// TIA Portal V18 export
ORGANIZATION_BLOCK "Safety"   // OB126, LAD, ProgramCycle
TITLE = "Main Program Sweep (Cycle)"
{ S7_Optimized_Access := 'TRUE' }
VERSION : 0.1
// stored: AutoNumber true, IsIECCheckEnabled false, SetENOAutomatically false
   VAR_INPUT
      Initial_Call : Bool;   // Initial call of this OB
      Remanence : Bool;   // =True, if remanent data are available
   END_VAR
   VAR_TEMP
      FaultReset : Bool;
      bRetVal : Int;
   END_VAR
   VAR_TEMP   // added for the SCL form of the ladder/FBD networks
      _w1 : Bool;
      _w2 : Bool;
      _w3 : Bool;
   END_VAR
BEGIN

REGION Network 1: ESTOP Release Edge
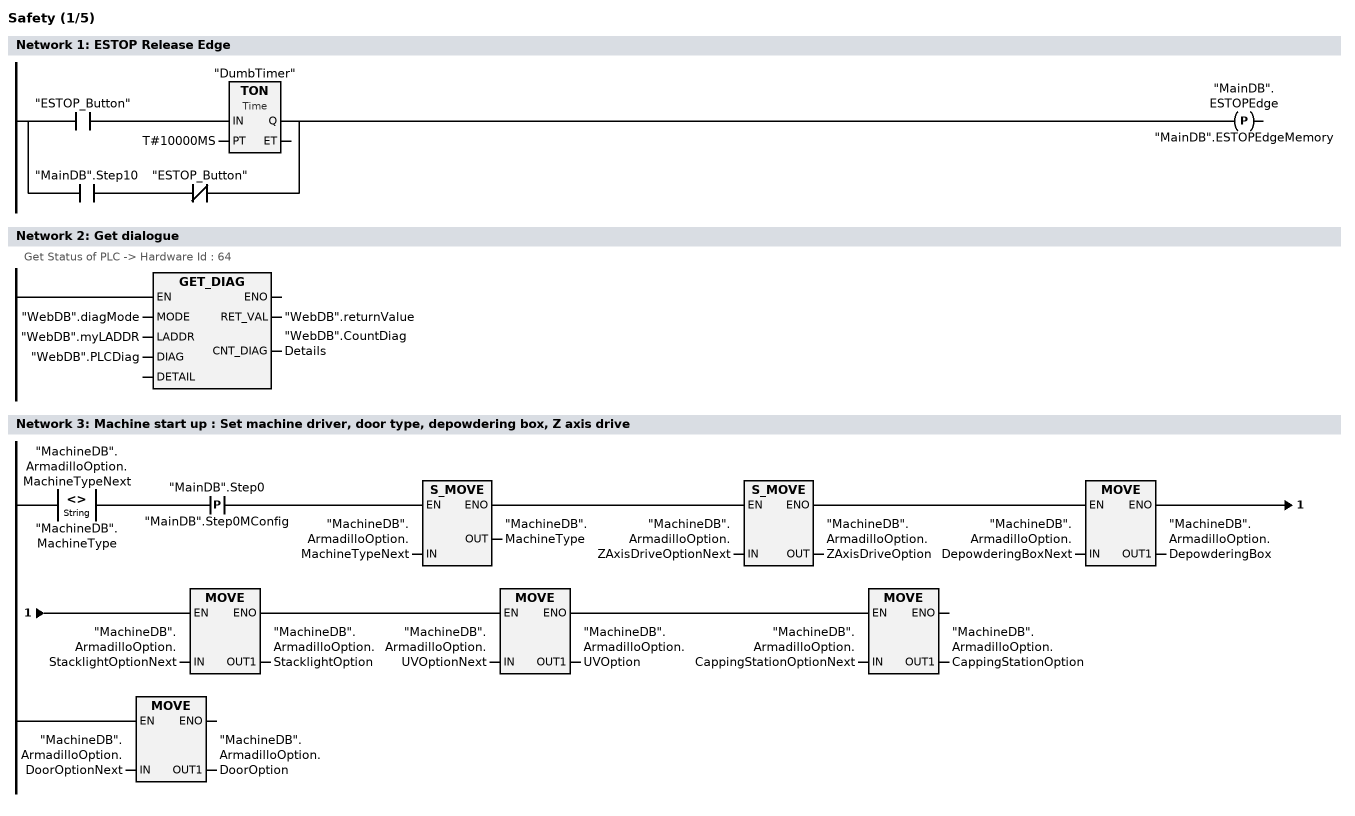
   "DumbTimer".TON(IN := "ESTOP_Button", PT := T#10000MS);
   #_w1 := "DumbTimer".Q OR ("MainDB".Step10 AND NOT "ESTOP_Button");
   "MainDB".ESTOPEdge := #_w1 AND NOT "MainDB".ESTOPEdgeMemory;   // rising edge
   "MainDB".ESTOPEdgeMemory := #_w1;
END_REGION

REGION Network 2: Get dialogue
   // Get Status of PLC -> Hardware Id : 64
   RUNG wire#powerrail
      GET_DIAG(MODE := "WebDB".diagMode, LADDR := "WebDB".myLADDR, DIAG := "WebDB".PLCDiag, DETAIL :=, RET_VAL => "WebDB".returnValue, CNT_DIAG => "WebDB".CountDiagDetails)
   END_RUNG
   // the same network as SCL:
   "WebDB".returnValue := GET_DIAG(MODE := "WebDB".diagMode,
                           LADDR := "WebDB".myLADDR,
                           DIAG := "WebDB".PLCDiag,
                           CNT_DIAG => "WebDB".CountDiagDetails);
END_REGION

REGION Network 3: Machine start up : Set machine driver, door type, depowdering box, Z axis drive
   RUNG wire#powerrail
      { S7_Templates := "SrcType := String" } NE_Contact(in1 := "MachineDB".ArmadilloOption.MachineTypeNext, in2 := "MachineDB".MachineType)
      P_Contact(operand := "MainDB".Step0, bit := "MainDB".Step0MConfig)
      S_Move(in := "MachineDB".ArmadilloOption.MachineTypeNext, out => "MachineDB".MachineType)
      S_Move(in := "MachineDB".ArmadilloOption.ZAxisDriveOptionNext, out => "MachineDB".ArmadilloOption.ZAxisDriveOption)
      Move(in := "MachineDB".ArmadilloOption.DepowderingBoxNext, out1 => "MachineDB".ArmadilloOption.DepowderingBox)
      Move(in := "MachineDB".ArmadilloOption.StacklightOptionNext, out1 => "MachineDB".ArmadilloOption.StacklightOption)
      Move(in := "MachineDB".ArmadilloOption.UVOptionNext, out1 => "MachineDB".ArmadilloOption.UVOption)
      Move(in := "MachineDB".ArmadilloOption.CappingStationOptionNext, out1 => "MachineDB".ArmadilloOption.CappingStationOption)
   END_RUNG
   RUNG wire#powerrail
      Move(in := "MachineDB".ArmadilloOption.DoorOptionNext, out1 => "MachineDB".ArmadilloOption.DoorOption)
   END_RUNG
   // the same network as SCL:
   #_w1 := ("MachineDB".ArmadilloOption.MachineTypeNext <> "MachineDB".MachineType) AND "MainDB".Step0 AND NOT "MainDB".Step0MConfig;   // rising edge of "MainDB".Step0
   "MainDB".Step0MConfig := "MainDB".Step0;
   IF #_w1 THEN
       "MachineDB".MachineType := "MachineDB".ArmadilloOption.MachineTypeNext;
       "MachineDB".ArmadilloOption.ZAxisDriveOption := "MachineDB".ArmadilloOption.ZAxisDriveOptionNext;
       "MachineDB".ArmadilloOption.DepowderingBox := "MachineDB".ArmadilloOption.DepowderingBoxNext;
       "MachineDB".ArmadilloOption.StacklightOption := "MachineDB".ArmadilloOption.StacklightOptionNext;
       "MachineDB".ArmadilloOption.UVOption := "MachineDB".ArmadilloOption.UVOptionNext;
       "MachineDB".ArmadilloOption.CappingStationOption := "MachineDB".ArmadilloOption.CappingStationOptionNext;
   END_IF;
   "MachineDB".ArmadilloOption.DoorOption := "MachineDB".ArmadilloOption.DoorOptionNext;
END_REGION

REGION Network 4: MachineDriverSettingArray
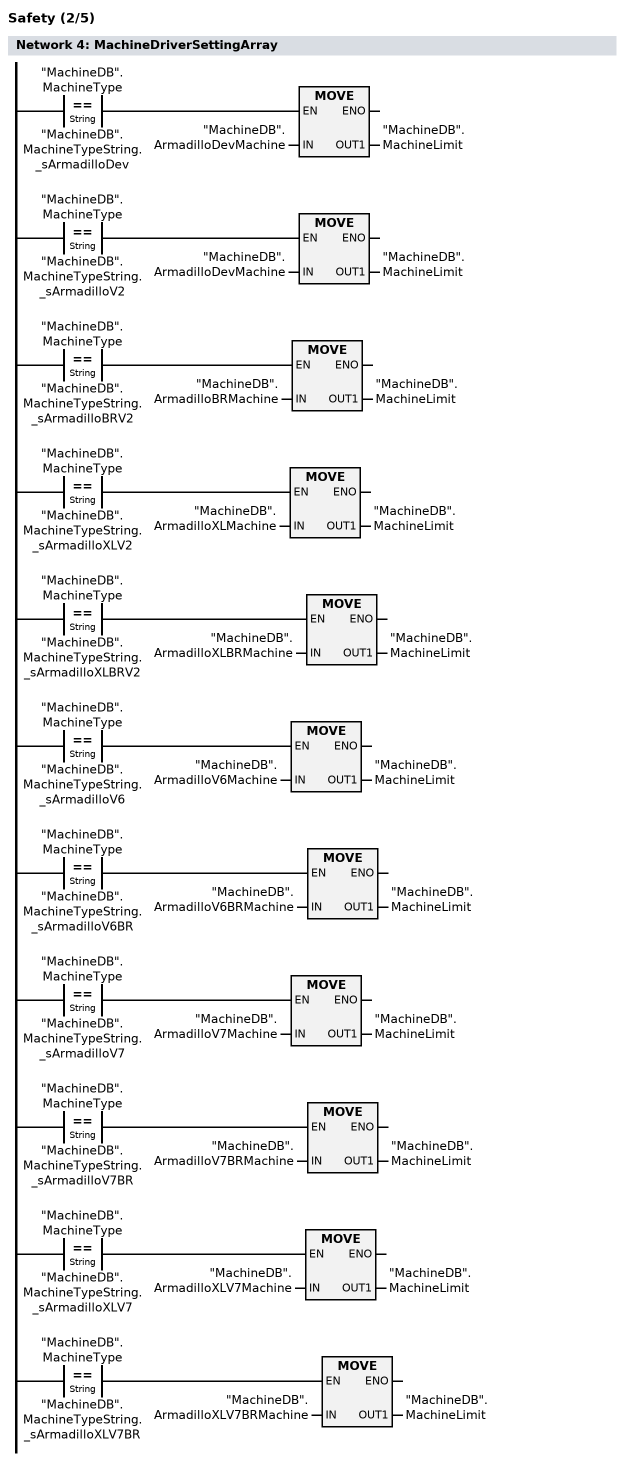
   RUNG wire#powerrail
      { S7_Templates := "SrcType := String" } EQ_Contact(in1 := "MachineDB".MachineType, in2 := "MachineDB".MachineTypeString._sArmadilloDev)
      Move(in := "MachineDB".ArmadilloDevMachine, out1 => "MachineDB".MachineLimit)
   END_RUNG
   RUNG wire#powerrail
      { S7_Templates := "SrcType := String" } EQ_Contact(in1 := "MachineDB".MachineType, in2 := "MachineDB".MachineTypeString._sArmadilloV2)
      Move(in := "MachineDB".ArmadilloDevMachine, out1 => "MachineDB".MachineLimit)
   END_RUNG
   RUNG wire#powerrail
      { S7_Templates := "SrcType := String" } EQ_Contact(in1 := "MachineDB".MachineType, in2 := "MachineDB".MachineTypeString._sArmadilloBRV2)
      Move(in := "MachineDB".ArmadilloBRMachine, out1 => "MachineDB".MachineLimit)
   END_RUNG
   RUNG wire#powerrail
      { S7_Templates := "SrcType := String" } EQ_Contact(in1 := "MachineDB".MachineType, in2 := "MachineDB".MachineTypeString._sArmadilloXLV2)
      Move(in := "MachineDB".ArmadilloXLMachine, out1 => "MachineDB".MachineLimit)
   END_RUNG
   RUNG wire#powerrail
      { S7_Templates := "SrcType := String" } EQ_Contact(in1 := "MachineDB".MachineType, in2 := "MachineDB".MachineTypeString._sArmadilloXLBRV2)
      Move(in := "MachineDB".ArmadilloXLBRMachine, out1 => "MachineDB".MachineLimit)
   END_RUNG
   RUNG wire#powerrail
      { S7_Templates := "SrcType := String" } EQ_Contact(in1 := "MachineDB".MachineType, in2 := "MachineDB".MachineTypeString._sArmadilloV6)
      Move(in := "MachineDB".ArmadilloV6Machine, out1 => "MachineDB".MachineLimit)
   END_RUNG
   RUNG wire#powerrail
      { S7_Templates := "SrcType := String" } EQ_Contact(in1 := "MachineDB".MachineType, in2 := "MachineDB".MachineTypeString._sArmadilloV6BR)
      Move(in := "MachineDB".ArmadilloV6BRMachine, out1 => "MachineDB".MachineLimit)
   END_RUNG
   RUNG wire#powerrail
      { S7_Templates := "SrcType := String" } EQ_Contact(in1 := "MachineDB".MachineType, in2 := "MachineDB".MachineTypeString._sArmadilloV7)
      Move(in := "MachineDB".ArmadilloV7Machine, out1 => "MachineDB".MachineLimit)
   END_RUNG
   RUNG wire#powerrail
      { S7_Templates := "SrcType := String" } EQ_Contact(in1 := "MachineDB".MachineType, in2 := "MachineDB".MachineTypeString._sArmadilloV7BR)
      Move(in := "MachineDB".ArmadilloV7BRMachine, out1 => "MachineDB".MachineLimit)
   END_RUNG
   RUNG wire#powerrail
      { S7_Templates := "SrcType := String" } EQ_Contact(in1 := "MachineDB".MachineType, in2 := "MachineDB".MachineTypeString._sArmadilloXLV7)
      Move(in := "MachineDB".ArmadilloXLV7Machine, out1 => "MachineDB".MachineLimit)
   END_RUNG
   RUNG wire#powerrail
      { S7_Templates := "SrcType := String" } EQ_Contact(in1 := "MachineDB".MachineType, in2 := "MachineDB".MachineTypeString._sArmadilloXLV7BR)
      Move(in := "MachineDB".ArmadilloXLV7BRMachine, out1 => "MachineDB".MachineLimit)
   END_RUNG
   // the same network as SCL:
   IF "MachineDB".MachineType = "MachineDB".MachineTypeString._sArmadilloDev THEN
       "MachineDB".MachineLimit := "MachineDB".ArmadilloDevMachine;
   END_IF;
   IF "MachineDB".MachineType = "MachineDB".MachineTypeString._sArmadilloV2 THEN
       "MachineDB".MachineLimit := "MachineDB".ArmadilloDevMachine;
   END_IF;
   IF "MachineDB".MachineType = "MachineDB".MachineTypeString._sArmadilloBRV2 THEN
       "MachineDB".MachineLimit := "MachineDB".ArmadilloBRMachine;
   END_IF;
   IF "MachineDB".MachineType = "MachineDB".MachineTypeString._sArmadilloXLV2 THEN
       "MachineDB".MachineLimit := "MachineDB".ArmadilloXLMachine;
   END_IF;
   IF "MachineDB".MachineType = "MachineDB".MachineTypeString._sArmadilloXLBRV2 THEN
       "MachineDB".MachineLimit := "MachineDB".ArmadilloXLBRMachine;
   END_IF;
   IF "MachineDB".MachineType = "MachineDB".MachineTypeString._sArmadilloV6 THEN
       "MachineDB".MachineLimit := "MachineDB".ArmadilloV6Machine;
   END_IF;
   IF "MachineDB".MachineType = "MachineDB".MachineTypeString._sArmadilloV6BR THEN
       "MachineDB".MachineLimit := "MachineDB".ArmadilloV6BRMachine;
   END_IF;
   IF "MachineDB".MachineType = "MachineDB".MachineTypeString._sArmadilloV7 THEN
       "MachineDB".MachineLimit := "MachineDB".ArmadilloV7Machine;
   END_IF;
   IF "MachineDB".MachineType = "MachineDB".MachineTypeString._sArmadilloV7BR THEN
       "MachineDB".MachineLimit := "MachineDB".ArmadilloV7BRMachine;
   END_IF;
   IF "MachineDB".MachineType = "MachineDB".MachineTypeString._sArmadilloXLV7 THEN
       "MachineDB".MachineLimit := "MachineDB".ArmadilloXLV7Machine;
   END_IF;
   IF "MachineDB".MachineType = "MachineDB".MachineTypeString._sArmadilloXLV7BR THEN
       "MachineDB".MachineLimit := "MachineDB".ArmadilloXLV7BRMachine;
   END_IF;
END_REGION

REGION Network 5: No Go Zone 01
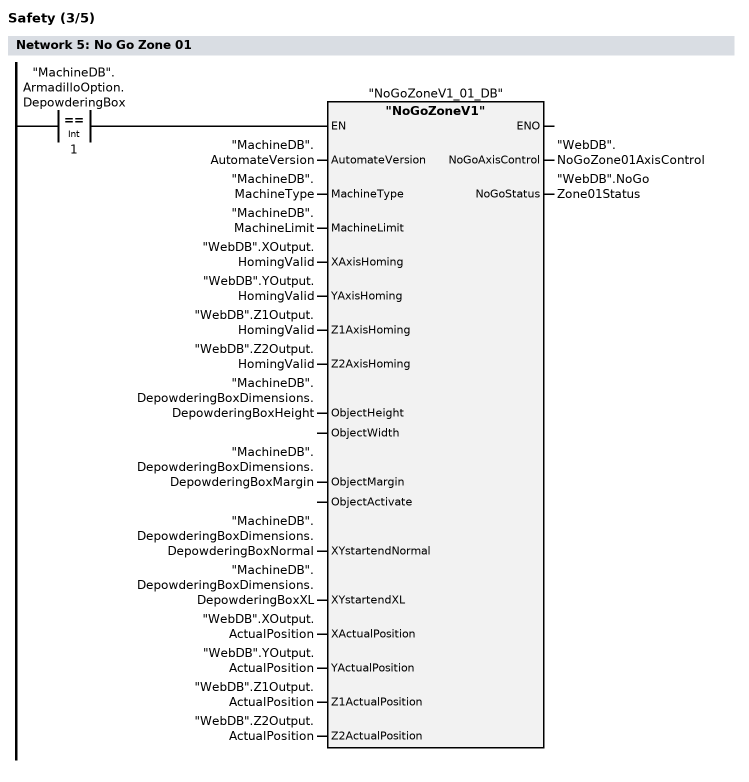
   RUNG wire#powerrail
      { S7_Templates := "SrcType := Int" } EQ_Contact(in1 := "MachineDB".ArmadilloOption.DepowderingBox, in2 := 1)
      "NoGoZoneV1_01_DB"(AutomateVersion := "MachineDB".AutomateVersion, MachineType := "MachineDB".MachineType, MachineLimit := "MachineDB".MachineLimit, XAxisHoming := "WebDB".XOutput.HomingValid, YAxisHoming := "WebDB".YOutput.HomingValid, Z1AxisHoming := "WebDB".Z1Output.HomingValid, Z2AxisHoming := "WebDB".Z2Output.HomingValid, ObjectHeight := "MachineDB".DepowderingBoxDimensions.DepowderingBoxHeight, ObjectWidth :=, ObjectMargin := "MachineDB".DepowderingBoxDimensions.DepowderingBoxMargin, ObjectActivate :=, XYstartendNormal := "MachineDB".DepowderingBoxDimensions.DepowderingBoxNormal, XYstartendXL := "MachineDB".DepowderingBoxDimensions.DepowderingBoxXL, XActualPosition := "WebDB".XOutput.ActualPosition, YActualPosition := "WebDB".YOutput.ActualPosition, Z1ActualPosition := "WebDB".Z1Output.ActualPosition, Z2ActualPosition := "WebDB".Z2Output.ActualPosition, NoGoAxisControl => "WebDB".NoGoZone01AxisControl, NoGoStatus => "WebDB".NoGoZone01Status)
   END_RUNG
   // the same network as SCL:
   IF "MachineDB".ArmadilloOption.DepowderingBox = 1 THEN
       "NoGoZoneV1_01_DB"(AutomateVersion := "MachineDB".AutomateVersion,   // "NoGoZoneV1"
                          MachineType := "MachineDB".MachineType,
                          MachineLimit := "MachineDB".MachineLimit,
                          XAxisHoming := "WebDB".XOutput.HomingValid,
                          YAxisHoming := "WebDB".YOutput.HomingValid,
                          Z1AxisHoming := "WebDB".Z1Output.HomingValid,
                          Z2AxisHoming := "WebDB".Z2Output.HomingValid,
                          ObjectHeight := "MachineDB".DepowderingBoxDimensions.DepowderingBoxHeight,
                          ObjectMargin := "MachineDB".DepowderingBoxDimensions.DepowderingBoxMargin,
                          XYstartendNormal := "MachineDB".DepowderingBoxDimensions.DepowderingBoxNormal,
                          XYstartendXL := "MachineDB".DepowderingBoxDimensions.DepowderingBoxXL,
                          XActualPosition := "WebDB".XOutput.ActualPosition,
                          YActualPosition := "WebDB".YOutput.ActualPosition,
                          Z1ActualPosition := "WebDB".Z1Output.ActualPosition,
                          Z2ActualPosition := "WebDB".Z2Output.ActualPosition,
                          NoGoAxisControl => "WebDB".NoGoZone01AxisControl,
                          NoGoStatus => "WebDB".NoGoZone01Status);
   END_IF;
END_REGION

REGION Network 6: Door Sensor
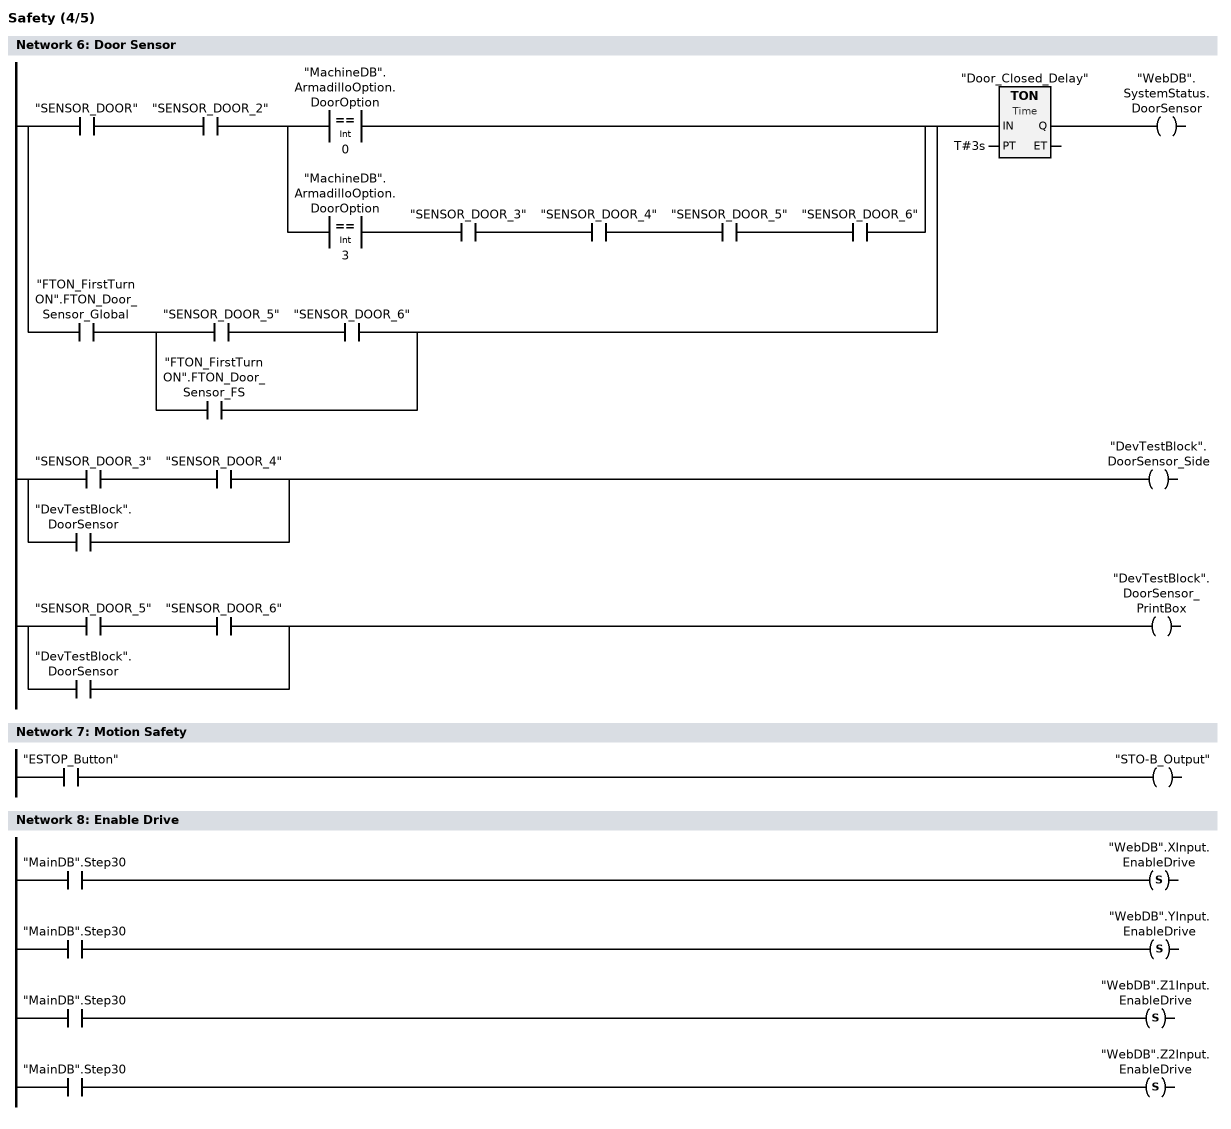
   RUNG wire#powerrail
      Contact( "SENSOR_DOOR" )
      Contact( "SENSOR_DOOR_2" )
      wire#w1
      { S7_Templates := "SrcType := Int" } EQ_Contact(in1 := "MachineDB".ArmadilloOption.DoorOption, in2 := 0)
      wire#w2
      { S7_Templates := "time_type := Time" } "Door_Closed_Delay".TON(pt := T#3s, et =>)
      Coil( "WebDB".SystemStatus.DoorSensor )
   END_RUNG
   RUNG wire#w1
      { S7_Templates := "SrcType := Int" } EQ_Contact(in1 := "MachineDB".ArmadilloOption.DoorOption, in2 := 3)
      Contact( "SENSOR_DOOR_3" )
      Contact( "SENSOR_DOOR_4" )
      Contact( "SENSOR_DOOR_5" )
      Contact( "SENSOR_DOOR_6" )
   END_RUNG wire#w2
   RUNG wire#powerrail
      Contact( "FTON_FirstTurnON".FTON_Door_Sensor_Global )
      wire#w3
      Contact( "SENSOR_DOOR_5" )
      Contact( "SENSOR_DOOR_6" )
   END_RUNG wire#w2
   RUNG wire#w3
      Contact( "FTON_FirstTurnON".FTON_Door_Sensor_FS )
   END_RUNG wire#w2
   RUNG wire#powerrail
      Contact( "SENSOR_DOOR_3" )
      Contact( "SENSOR_DOOR_4" )
      wire#w4
      Coil( "DevTestBlock".DoorSensor_Side )
   END_RUNG
   RUNG wire#powerrail
      Contact( "DevTestBlock".DoorSensor )
   END_RUNG wire#w4
   RUNG wire#powerrail
      Contact( "SENSOR_DOOR_5" )
      Contact( "SENSOR_DOOR_6" )
      wire#w5
      Coil( "DevTestBlock".DoorSensor_PrintBox )
   END_RUNG
   RUNG wire#powerrail
      Contact( "DevTestBlock".DoorSensor )
   END_RUNG wire#w5
   // the same network as SCL:
   "Door_Closed_Delay".TON(IN := ("SENSOR_DOOR" AND "SENSOR_DOOR_2" AND (("MachineDB".ArmadilloOption.DoorOption = 0) OR (("MachineDB".ArmadilloOption.DoorOption = 3) AND "SENSOR_DOOR_3" AND "SENSOR_DOOR_4" AND "SENSOR_DOOR_5" AND "SENSOR_DOOR_6"))) OR ("FTON_FirstTurnON".FTON_Door_Sensor_Global AND (("SENSOR_DOOR_5" AND "SENSOR_DOOR_6") OR "FTON_FirstTurnON".FTON_Door_Sensor_FS)),
                           PT := T#3s);
   "WebDB".SystemStatus.DoorSensor := "Door_Closed_Delay".Q;
   "DevTestBlock".DoorSensor_Side := ("SENSOR_DOOR_3" AND "SENSOR_DOOR_4") OR "DevTestBlock".DoorSensor;
   "DevTestBlock".DoorSensor_PrintBox := ("SENSOR_DOOR_5" AND "SENSOR_DOOR_6") OR "DevTestBlock".DoorSensor;
END_REGION

REGION Network 7: Motion Safety
   RUNG wire#powerrail
      Contact( "ESTOP_Button" )
      Coil( "STO-B_Output" )
   END_RUNG
   // the same network as SCL:
   "STO-B_Output" := "ESTOP_Button";
END_REGION

REGION Network 8: Enable Drive
   RUNG wire#powerrail
      Contact( "MainDB".Step30 )
      S_Coil( "WebDB".XInput.EnableDrive )
   END_RUNG
   RUNG wire#powerrail
      Contact( "MainDB".Step30 )
      S_Coil( "WebDB".YInput.EnableDrive )
   END_RUNG
   RUNG wire#powerrail
      Contact( "MainDB".Step30 )
      S_Coil( "WebDB".Z1Input.EnableDrive )
   END_RUNG
   RUNG wire#powerrail
      Contact( "MainDB".Step30 )
      S_Coil( "WebDB".Z2Input.EnableDrive )
   END_RUNG
   // the same network as SCL:
   IF "MainDB".Step30 THEN
       "WebDB".XInput.EnableDrive := TRUE;
       "WebDB".YInput.EnableDrive := TRUE;
       "WebDB".Z1Input.EnableDrive := TRUE;
       "WebDB".Z2Input.EnableDrive := TRUE;
   END_IF;
END_REGION

REGION Network 9: Disable Drive
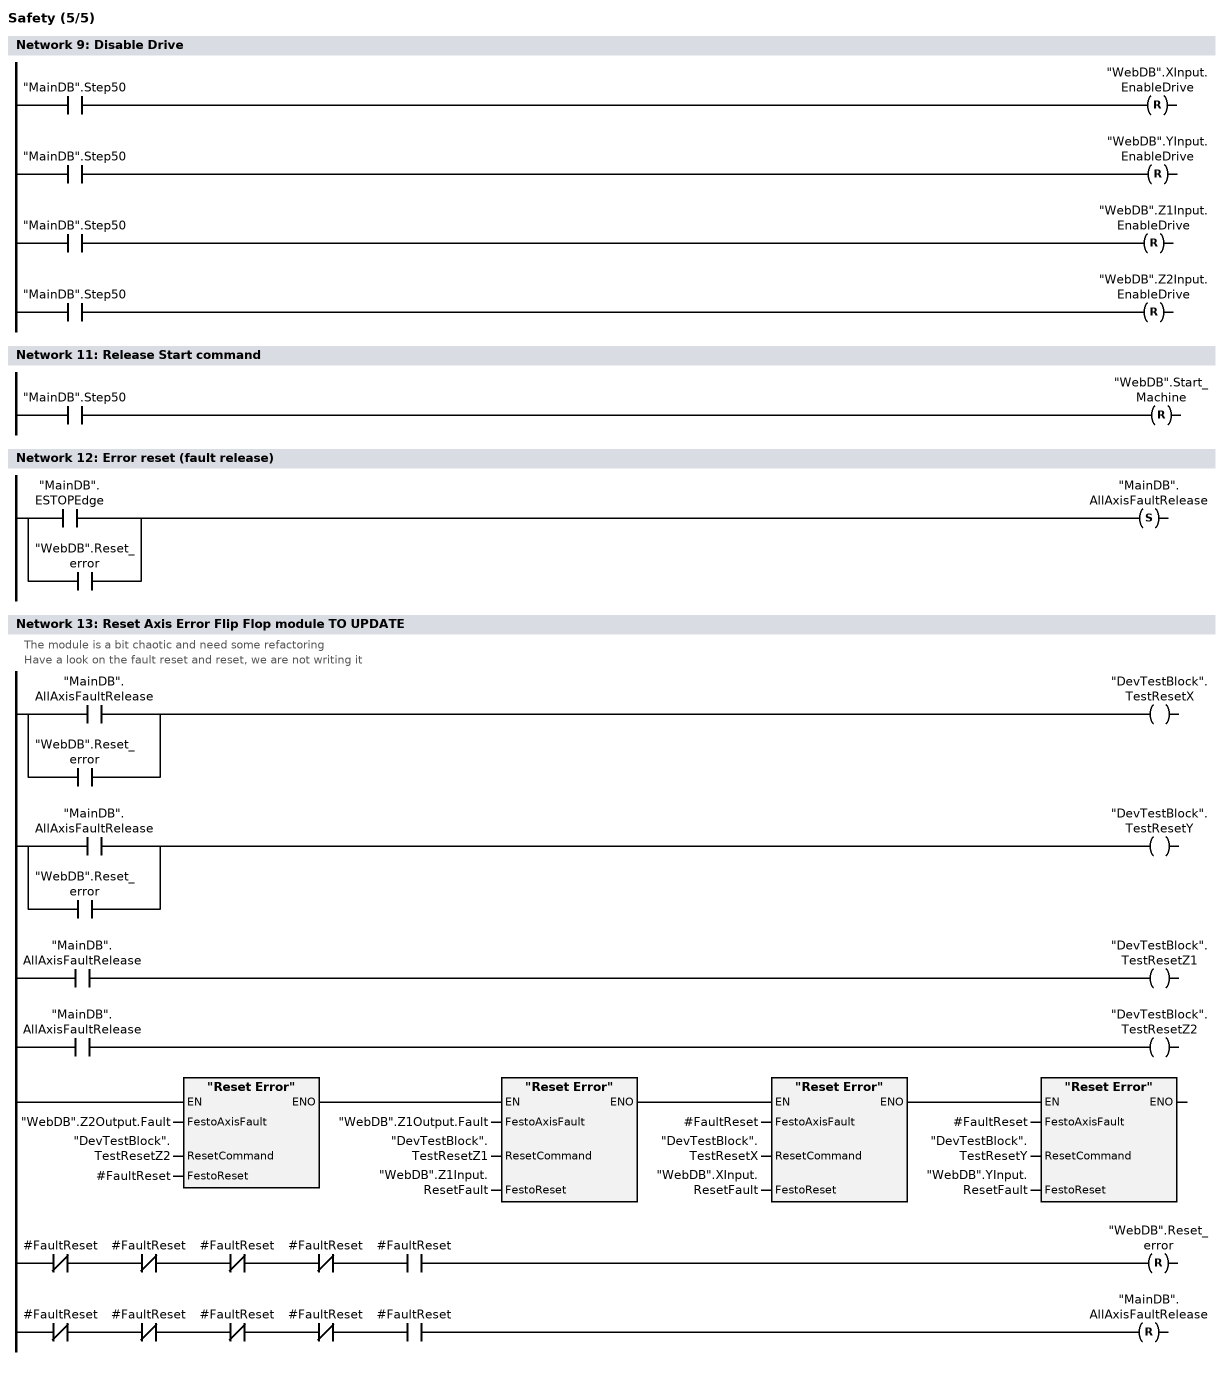
   RUNG wire#powerrail
      Contact( "MainDB".Step50 )
      R_Coil( "WebDB".XInput.EnableDrive )
   END_RUNG
   RUNG wire#powerrail
      Contact( "MainDB".Step50 )
      R_Coil( "WebDB".YInput.EnableDrive )
   END_RUNG
   RUNG wire#powerrail
      Contact( "MainDB".Step50 )
      R_Coil( "WebDB".Z1Input.EnableDrive )
   END_RUNG
   RUNG wire#powerrail
      Contact( "MainDB".Step50 )
      R_Coil( "WebDB".Z2Input.EnableDrive )
   END_RUNG
   // the same network as SCL:
   IF "MainDB".Step50 THEN
       "WebDB".XInput.EnableDrive := FALSE;
       "WebDB".YInput.EnableDrive := FALSE;
       "WebDB".Z1Input.EnableDrive := FALSE;
       "WebDB".Z2Input.EnableDrive := FALSE;
   END_IF;
END_REGION

REGION Network 10: Add Ons Safety
END_REGION

REGION Network 11: Release Start command
   RUNG wire#powerrail
      Contact( "MainDB".Step50 )
      R_Coil( "WebDB".Start_Machine )
   END_RUNG
   // the same network as SCL:
   IF "MainDB".Step50 THEN "WebDB".Start_Machine := FALSE; END_IF;
END_REGION

REGION Network 12: Error reset (fault release)
   RUNG wire#powerrail
      Contact( "MainDB".ESTOPEdge )
      wire#w1
      S_Coil( "MainDB".AllAxisFaultRelease )
   END_RUNG
   RUNG wire#powerrail
      Contact( "WebDB".Reset_error )
   END_RUNG wire#w1
   // the same network as SCL:
   IF "MainDB".ESTOPEdge OR "WebDB".Reset_error THEN "MainDB".AllAxisFaultRelease := TRUE; END_IF;
END_REGION

REGION Network 13: Reset Axis Error Flip Flop module TO UPDATE
   // The module is a bit chaotic and need some refactoring
   // Have a look on the fault reset and reset, we are not writing it
   RUNG wire#powerrail
      Contact( "MainDB".AllAxisFaultRelease )
      wire#w1
      Coil( "DevTestBlock".TestResetX )
   END_RUNG
   RUNG wire#powerrail
      Contact( "WebDB".Reset_error )
   END_RUNG wire#w1
   RUNG wire#powerrail
      Contact( "MainDB".AllAxisFaultRelease )
      wire#w2
      Coil( "DevTestBlock".TestResetY )
   END_RUNG
   RUNG wire#powerrail
      Contact( "WebDB".Reset_error )
   END_RUNG wire#w2
   RUNG wire#powerrail
      Contact( "MainDB".AllAxisFaultRelease )
      Coil( "DevTestBlock".TestResetZ1 )
   END_RUNG
   RUNG wire#powerrail
      Contact( "MainDB".AllAxisFaultRelease )
      Coil( "DevTestBlock".TestResetZ2 )
   END_RUNG
   RUNG wire#powerrail
      "Reset Error"(FestoAxisFault := "WebDB".Z2Output.Fault, ResetCommand := "DevTestBlock".TestResetZ2, FestoReset := #FaultReset)
      "Reset Error"(FestoAxisFault := "WebDB".Z1Output.Fault, ResetCommand := "DevTestBlock".TestResetZ1, FestoReset := "WebDB".Z1Input.ResetFault)
      "Reset Error"(FestoAxisFault := #FaultReset, ResetCommand := "DevTestBlock".TestResetX, FestoReset := "WebDB".XInput.ResetFault)
      "Reset Error"(FestoAxisFault := #FaultReset, ResetCommand := "DevTestBlock".TestResetY, FestoReset := "WebDB".YInput.ResetFault)
   END_RUNG
   RUNG wire#powerrail
      I_Contact( #FaultReset )
      I_Contact( #FaultReset )
      I_Contact( #FaultReset )
      I_Contact( #FaultReset )
      Contact( #FaultReset )
      R_Coil( "WebDB".Reset_error )
   END_RUNG
   RUNG wire#powerrail
      I_Contact( #FaultReset )
      I_Contact( #FaultReset )
      I_Contact( #FaultReset )
      I_Contact( #FaultReset )
      Contact( #FaultReset )
      R_Coil( "MainDB".AllAxisFaultRelease )
   END_RUNG
   // the same network as SCL:
   "DevTestBlock".TestResetX := "MainDB".AllAxisFaultRelease OR "WebDB".Reset_error;
   "DevTestBlock".TestResetY := "MainDB".AllAxisFaultRelease OR "WebDB".Reset_error;
   "DevTestBlock".TestResetZ1 := "MainDB".AllAxisFaultRelease;
   "DevTestBlock".TestResetZ2 := "MainDB".AllAxisFaultRelease;
   "Reset Error"(FestoAxisFault := "WebDB".Z2Output.Fault,
                 ResetCommand := "DevTestBlock".TestResetZ2,
                 FestoReset := #FaultReset,
                 ENO => #_w1);
   "Reset Error"(EN := #_w1,
                 FestoAxisFault := "WebDB".Z1Output.Fault,
                 ResetCommand := "DevTestBlock".TestResetZ1,
                 FestoReset := "WebDB".Z1Input.ResetFault,
                 ENO => #_w2);
   "Reset Error"(EN := #_w2,
                 FestoAxisFault := #FaultReset,
                 ResetCommand := "DevTestBlock".TestResetX,
                 FestoReset := "WebDB".XInput.ResetFault,
                 ENO => #_w3);
   IF #_w3 THEN
       "Reset Error"(FestoAxisFault := #FaultReset,
                     ResetCommand := "DevTestBlock".TestResetY,
                     FestoReset := "WebDB".YInput.ResetFault);
   END_IF;
   IF NOT #FaultReset AND NOT #FaultReset AND NOT #FaultReset AND NOT #FaultReset AND #FaultReset THEN
       "WebDB".Reset_error := FALSE;
       "MainDB".AllAxisFaultRelease := FALSE;
   END_IF;
END_REGION
END_ORGANIZATION_BLOCK
